DATA_BLOCK "NeuroPLC_MLP_Weights"
{ S7_Optimized_Access := 'FALSE' }
VERSION : 0.1
NON_RETAIN
   STRUCT
      w0 : ARRAY[0..895] OF REAL;  // W(32x28)
      b1 : ARRAY[0..31] OF REAL;  // bias(32)
      w2 : ARRAY[0..511] OF REAL;  // W(16x32)
      b3 : ARRAY[0..15] OF REAL;  // bias(16)
      w4 : ARRAY[0..63] OF REAL;  // W(4x16)
      b5 : ARRAY[0..3] OF REAL;  // bias(4)
   END_STRUCT;
BEGIN

      // MatMul 'fc0': W + bias
      w0[0] := 0.5694862; w0[1] := -0.0095692; w0[2] := 0.7619486; w0[3] := 0.2215109; w0[4] := -0.3561512; w0[5] := -0.2522623; w0[6] := 0.2582799; w0[7] := 0.0099258;
      w0[8] := 0.3836571; w0[9] := -0.0658457; w0[10] := 0.1010401; w0[11] := -0.2984352; w0[12] := 0.1934527; w0[13] := -0.2640140; w0[14] := 0.1362384; w0[15] := -0.0190728;
      w0[16] := -0.2375232; w0[17] := -0.1084833; w0[18] := -0.3846658; w0[19] := 0.3771667; w0[20] := -0.1136759; w0[21] := -0.1259104; w0[22] := -0.1682155; w0[23] := 0.4097499;
      w0[24] := -0.2194012; w0[25] := -0.2356472; w0[26] := -0.1771912; w0[27] := 0.1675407; w0[28] := 0.1454716; w0[29] := -0.3696787; w0[30] := -0.2783369; w0[31] := -0.1873165;
      w0[32] := 0.0781848; w0[33] := -0.3527579; w0[34] := -0.2131715; w0[35] := -0.4139680; w0[36] := -0.5927966; w0[37] := 0.3198802; w0[38] := -0.5640871; w0[39] := -0.2003005;
      w0[40] := 0.1832723; w0[41] := 0.2237836; w0[42] := 0.1929916; w0[43] := 0.2185234; w0[44] := 0.1214973; w0[45] := 0.0208249; w0[46] := 0.2776418; w0[47] := 0.6831574;
      w0[48] := -0.1655439; w0[49] := -0.2658227; w0[50] := -0.2709237; w0[51] := 0.0986710; w0[52] := 0.1128972; w0[53] := -0.2047481; w0[54] := -0.3872808; w0[55] := 0.1596099;
      w0[56] := -0.2523361; w0[57] := 0.2758174; w0[58] := 0.2686562; w0[59] := -0.5177624; w0[60] := -0.1129441; w0[61] := -0.2192100; w0[62] := 0.3343761; w0[63] := -0.0422801;
      w0[64] := -0.3068857; w0[65] := 0.2210509; w0[66] := -0.5496964; w0[67] := 0.3709493; w0[68] := 0.0747587; w0[69] := -0.1170707; w0[70] := -0.3195110; w0[71] := 0.0277475;
      w0[72] := -0.2577946; w0[73] := 0.0641775; w0[74] := 0.2055912; w0[75] := 0.6039576; w0[76] := -0.5010191; w0[77] := 0.0377836; w0[78] := 0.2038942; w0[79] := -0.0376425;
      w0[80] := 0.1546009; w0[81] := 0.3260912; w0[82] := -0.1506072; w0[83] := 0.0569262; w0[84] := -0.1928782; w0[85] := -0.1984540; w0[86] := -0.0539345; w0[87] := 0.3094364;
      w0[88] := 0.2289592; w0[89] := -0.4250050; w0[90] := -0.0399776; w0[91] := 0.0658291; w0[92] := 0.2534966; w0[93] := -0.0973715; w0[94] := -0.3647969; w0[95] := -0.0156060;
      w0[96] := -0.5209337; w0[97] := 0.2564455; w0[98] := 0.1338747; w0[99] := 0.3502659; w0[100] := -0.3756513; w0[101] := 0.2530890; w0[102] := 0.0984663; w0[103] := 0.6602526;
      w0[104] := 0.3365156; w0[105] := -0.2521311; w0[106] := 0.0946512; w0[107] := -0.6085349; w0[108] := -0.5372492; w0[109] := 0.0455726; w0[110] := -0.0786947; w0[111] := 0.0370381;
      w0[112] := -0.5858350; w0[113] := -0.7779619; w0[114] := -0.7385424; w0[115] := -0.2071060; w0[116] := 0.2831336; w0[117] := 0.3243212; w0[118] := 0.2366221; w0[119] := -0.2105746;
      w0[120] := -0.3834608; w0[121] := -0.6828474; w0[122] := 0.1007835; w0[123] := 0.0381121; w0[124] := 0.3126857; w0[125] := 0.0975034; w0[126] := 0.0499541; w0[127] := -0.0530838;
      w0[128] := 0.0799674; w0[129] := -0.1505451; w0[130] := -0.4892448; w0[131] := -0.3954702; w0[132] := 0.1594549; w0[133] := 0.2307071; w0[134] := -0.0041823; w0[135] := 0.5944483;
      w0[136] := -0.2759206; w0[137] := -0.4257804; w0[138] := -0.3279784; w0[139] := -0.2977980; w0[140] := 0.0038754; w0[141] := 0.3761657; w0[142] := 0.4177073; w0[143] := 0.0741864;
      w0[144] := 0.3750937; w0[145] := 0.2039272; w0[146] := -0.2429399; w0[147] := -0.3849822; w0[148] := 0.1600508; w0[149] := -0.1581226; w0[150] := -0.0233814; w0[151] := -0.1151747;
      w0[152] := -0.5731639; w0[153] := -0.0274457; w0[154] := 0.1195597; w0[155] := -0.2395748; w0[156] := 0.2293357; w0[157] := -0.0251415; w0[158] := 0.3937997; w0[159] := -0.1454628;
      w0[160] := -0.0673693; w0[161] := 0.2948158; w0[162] := 0.5630679; w0[163] := -0.3092144; w0[164] := 0.1832785; w0[165] := 0.0043120; w0[166] := 0.0011036; w0[167] := 0.2549984;
      w0[168] := 0.1242365; w0[169] := -0.1573328; w0[170] := 0.1472307; w0[171] := 0.2971004; w0[172] := 0.1052006; w0[173] := 0.3616425; w0[174] := -0.1347494; w0[175] := -0.3794992;
      w0[176] := 0.5467421; w0[177] := -0.1476457; w0[178] := 0.3496484; w0[179] := -0.0583753; w0[180] := 0.2853532; w0[181] := -0.3058073; w0[182] := -0.1615329; w0[183] := -0.5229150;
      w0[184] := 0.2140338; w0[185] := -0.2294949; w0[186] := 0.2921923; w0[187] := 0.0373898; w0[188] := 0.3493846; w0[189] := 0.5938788; w0[190] := 0.0955027; w0[191] := -0.1719695;
      w0[192] := 0.6582399; w0[193] := -0.4911650; w0[194] := 0.1269870; w0[195] := -0.4129370; w0[196] := -0.2735490; w0[197] := -0.2155660; w0[198] := 0.4269275; w0[199] := -0.1273027;
      w0[200] := -0.2414422; w0[201] := -0.3611139; w0[202] := 0.6480063; w0[203] := 0.3808921; w0[204] := -0.2189153; w0[205] := 0.0094489; w0[206] := 0.6784652; w0[207] := 0.3757944;
      w0[208] := 0.5965886; w0[209] := 0.3704935; w0[210] := 0.3205929; w0[211] := 0.2190031; w0[212] := -0.3913886; w0[213] := 0.2046225; w0[214] := 0.7660633; w0[215] := 0.5648795;
      w0[216] := 0.0447379; w0[217] := -0.1363681; w0[218] := -0.1653181; w0[219] := -0.3211187; w0[220] := 0.0557173; w0[221] := -0.6775630; w0[222] := 0.2077208; w0[223] := 0.1863764;
      w0[224] := 0.0122372; w0[225] := -0.1510706; w0[226] := -0.0393031; w0[227] := -0.2373850; w0[228] := 0.3297745; w0[229] := -0.3327326; w0[230] := -0.1183226; w0[231] := 0.3871697;
      w0[232] := -0.4481050; w0[233] := -0.2065133; w0[234] := 0.1012533; w0[235] := -0.2578072; w0[236] := 0.0634624; w0[237] := -0.1246978; w0[238] := 0.1465549; w0[239] := -0.5023389;
      w0[240] := 0.0640146; w0[241] := 0.1963426; w0[242] := 0.6648222; w0[243] := -0.6102669; w0[244] := -0.2871900; w0[245] := -0.3684005; w0[246] := -0.4533643; w0[247] := -0.1819637;
      w0[248] := -0.3802012; w0[249] := 0.4682154; w0[250] := 0.1991423; w0[251] := 0.5698866; w0[252] := 0.3063245; w0[253] := 0.1672625; w0[254] := 0.2611240; w0[255] := -0.6845852;
      w0[256] := -0.1005014; w0[257] := -0.6641653; w0[258] := -0.2544510; w0[259] := 0.1954752; w0[260] := -0.2994281; w0[261] := 0.3571715; w0[262] := -0.0372742; w0[263] := -0.0310561;
      w0[264] := 0.1959654; w0[265] := -0.1060541; w0[266] := 0.3827632; w0[267] := -0.3923316; w0[268] := -0.5924090; w0[269] := 0.0670658; w0[270] := 0.3532278; w0[271] := 0.6439264;
      w0[272] := 0.1193878; w0[273] := -0.5490641; w0[274] := -0.6517076; w0[275] := 0.2266813; w0[276] := 0.2735080; w0[277] := 0.2562127; w0[278] := 0.3711089; w0[279] := -0.0201157;
      w0[280] := 0.5907255; w0[281] := 0.3026478; w0[282] := 0.0879490; w0[283] := -0.1103418; w0[284] := 0.0830003; w0[285] := 0.0901832; w0[286] := 0.4872787; w0[287] := -0.4248994;
      w0[288] := 0.6916616; w0[289] := 0.0068263; w0[290] := 0.0377772; w0[291] := -0.3450460; w0[292] := 0.5848706; w0[293] := -0.0756037; w0[294] := 0.0390328; w0[295] := -0.4139087;
      w0[296] := -0.1527735; w0[297] := -0.2285863; w0[298] := 0.3310088; w0[299] := 0.2031009; w0[300] := -0.5309294; w0[301] := -0.4607368; w0[302] := 0.1824918; w0[303] := -0.1911459;
      w0[304] := -0.1732452; w0[305] := -0.3283744; w0[306] := -0.0425148; w0[307] := -0.0754750; w0[308] := -0.0751830; w0[309] := -0.0057766; w0[310] := -0.0669558; w0[311] := -0.0518108;
      w0[312] := -0.1100485; w0[313] := 0.4202482; w0[314] := 0.1722786; w0[315] := 0.2540640; w0[316] := -0.2125306; w0[317] := -0.3108644; w0[318] := -0.1653187; w0[319] := 0.0082027;
      w0[320] := 0.1613134; w0[321] := 0.5696448; w0[322] := 0.4734836; w0[323] := -0.1820288; w0[324] := -0.0202256; w0[325] := 0.2319008; w0[326] := 0.6178575; w0[327] := -0.1729726;
      w0[328] := -0.5705087; w0[329] := -0.4175466; w0[330] := -0.0846097; w0[331] := -0.4305633; w0[332] := -0.0297265; w0[333] := -0.2146564; w0[334] := -0.0228577; w0[335] := 0.4386194;
      w0[336] := 0.1366172; w0[337] := 0.1275948; w0[338] := 0.2872518; w0[339] := -0.0469490; w0[340] := -0.3430789; w0[341] := -0.2333279; w0[342] := -0.0942715; w0[343] := -0.6695372;
      w0[344] := 0.3036573; w0[345] := 0.6706407; w0[346] := 0.4867018; w0[347] := 0.2229243; w0[348] := 0.1479198; w0[349] := 0.4786703; w0[350] := -0.1235309; w0[351] := -0.1444162;
      w0[352] := -0.1594525; w0[353] := 0.0118241; w0[354] := 0.3302614; w0[355] := 0.4612524; w0[356] := -0.1728074; w0[357] := -0.4940682; w0[358] := 0.2663130; w0[359] := 0.4213447;
      w0[360] := 0.1559720; w0[361] := 0.0927116; w0[362] := 0.2581408; w0[363] := 0.1484697; w0[364] := 0.5596921; w0[365] := 0.6450443; w0[366] := 0.2316463; w0[367] := -0.3064318;
      w0[368] := 0.3154030; w0[369] := 0.2504337; w0[370] := 0.2270162; w0[371] := -0.2362736; w0[372] := -0.1822204; w0[373] := 0.7585521; w0[374] := 0.2454521; w0[375] := -0.3572387;
      w0[376] := 0.1800293; w0[377] := 0.1965537; w0[378] := 0.1946464; w0[379] := 0.1738928; w0[380] := -0.1159788; w0[381] := -0.1791228; w0[382] := 0.3109314; w0[383] := 0.1039406;
      w0[384] := -0.2558490; w0[385] := -0.4132357; w0[386] := -0.1826324; w0[387] := -0.0949509; w0[388] := 0.0754630; w0[389] := -0.4951166; w0[390] := -0.0366096; w0[391] := -0.5241205;
      w0[392] := 0.0701182; w0[393] := 0.5458165; w0[394] := -0.3082272; w0[395] := -0.1620290; w0[396] := 0.2685293; w0[397] := -0.1115321; w0[398] := 0.5528188; w0[399] := 0.1818966;
      w0[400] := -0.2705870; w0[401] := -0.4477837; w0[402] := -0.3260813; w0[403] := -0.1751753; w0[404] := 0.3439055; w0[405] := 0.3690660; w0[406] := -0.0775537; w0[407] := -0.3291571;
      w0[408] := 0.3966570; w0[409] := 0.3747428; w0[410] := 0.2037812; w0[411] := 0.5063270; w0[412] := -0.0363616; w0[413] := -0.0945516; w0[414] := -0.2667596; w0[415] := -0.1880456;
      w0[416] := 0.2148547; w0[417] := -0.6592890; w0[418] := -0.2238534; w0[419] := -0.2862469; w0[420] := -0.8308039; w0[421] := -0.4430834; w0[422] := -0.0302747; w0[423] := 0.0918460;
      w0[424] := -0.3334551; w0[425] := -0.1804388; w0[426] := -0.1097601; w0[427] := 0.3427432; w0[428] := 0.0736062; w0[429] := -0.6790179; w0[430] := -0.2430520; w0[431] := -0.2084594;
      w0[432] := 0.1491454; w0[433] := -0.0083196; w0[434] := 0.2553293; w0[435] := 0.1678275; w0[436] := 0.0936099; w0[437] := 0.1736043; w0[438] := -0.5376837; w0[439] := -0.4510113;
      w0[440] := -0.3174161; w0[441] := 0.2371299; w0[442] := 0.3883051; w0[443] := 0.3464468; w0[444] := 0.1098732; w0[445] := 0.0205052; w0[446] := -0.2641115; w0[447] := -0.3012585;
      w0[448] := -0.5463231; w0[449] := -0.0684724; w0[450] := -0.1422806; w0[451] := -0.2644515; w0[452] := -0.4767578; w0[453] := -0.4182616; w0[454] := -0.4673964; w0[455] := -0.0129319;
      w0[456] := -0.5374129; w0[457] := -0.1050398; w0[458] := 0.0632549; w0[459] := 0.0568505; w0[460] := 0.2111508; w0[461] := 0.3917949; w0[462] := -0.0330271; w0[463] := 0.2814879;
      w0[464] := -0.3214771; w0[465] := 0.3430510; w0[466] := -0.3870021; w0[467] := -0.4042188; w0[468] := 0.1747253; w0[469] := 0.3262924; w0[470] := 0.5594077; w0[471] := 0.0277393;
      w0[472] := -0.2604083; w0[473] := 0.0503597; w0[474] := 0.3725081; w0[475] := -0.0544451; w0[476] := 0.0951887; w0[477] := -0.5271522; w0[478] := -0.3720489; w0[479] := 0.0333015;
      w0[480] := 0.3407656; w0[481] := -0.0524092; w0[482] := -0.3947720; w0[483] := 0.0632993; w0[484] := -0.4918242; w0[485] := -0.0408889; w0[486] := 0.5603451; w0[487] := 0.3429145;
      w0[488] := -0.0672607; w0[489] := -0.3218429; w0[490] := -0.3621323; w0[491] := -0.5524946; w0[492] := 0.3105496; w0[493] := 0.3352183; w0[494] := -0.6259544; w0[495] := -0.1107638;
      w0[496] := 0.0901521; w0[497] := 0.0038500; w0[498] := 0.5420415; w0[499] := 0.2380718; w0[500] := -0.0511688; w0[501] := -0.0771460; w0[502] := -0.0791493; w0[503] := -0.1069665;
      w0[504] := 0.6399192; w0[505] := -0.0014034; w0[506] := 0.3290343; w0[507] := -0.3565734; w0[508] := 0.2305476; w0[509] := -0.0417552; w0[510] := 0.2942790; w0[511] := -0.1355964;
      w0[512] := 0.0557771; w0[513] := 0.3271682; w0[514] := -0.3025698; w0[515] := 0.2897500; w0[516] := 0.1278277; w0[517] := -0.1560617; w0[518] := 0.2582703; w0[519] := -0.0549245;
      w0[520] := -0.0921321; w0[521] := 0.4996554; w0[522] := 0.0836308; w0[523] := 0.2032579; w0[524] := -0.1741465; w0[525] := -0.2436171; w0[526] := -0.3661414; w0[527] := -0.2924559;
      w0[528] := -0.4407195; w0[529] := 0.2304931; w0[530] := -0.2509898; w0[531] := -0.6881460; w0[532] := 0.1500384; w0[533] := 0.4429501; w0[534] := 0.5444623; w0[535] := 0.0644146;
      w0[536] := 0.1564979; w0[537] := 0.1936211; w0[538] := -0.2217757; w0[539] := 0.1632960; w0[540] := 0.0949209; w0[541] := 0.5449093; w0[542] := 0.3260632; w0[543] := 0.4177442;
      w0[544] := -0.1678705; w0[545] := -0.4614883; w0[546] := -0.1780888; w0[547] := 0.0282706; w0[548] := -0.3548764; w0[549] := 0.1119965; w0[550] := -0.6278588; w0[551] := -0.2857478;
      w0[552] := 0.3291071; w0[553] := -0.2958602; w0[554] := -0.2171935; w0[555] := 0.0488607; w0[556] := -0.2721503; w0[557] := -0.0109805; w0[558] := -0.2872001; w0[559] := -0.3800366;
      w0[560] := 0.7377275; w0[561] := 0.5175216; w0[562] := 0.4534726; w0[563] := 0.2131705; w0[564] := 0.1694544; w0[565] := 0.1088488; w0[566] := 0.2956495; w0[567] := -0.1219863;
      w0[568] := 0.4281839; w0[569] := 0.0482728; w0[570] := 0.3261450; w0[571] := 0.0147065; w0[572] := 0.0197347; w0[573] := -0.2837075; w0[574] := -0.2223815; w0[575] := -0.3011971;
      w0[576] := 0.4010099; w0[577] := 0.3606303; w0[578] := 0.5675586; w0[579] := -0.1933776; w0[580] := 0.1411208; w0[581] := 0.4412328; w0[582] := -0.3157989; w0[583] := 0.0737199;
      w0[584] := 0.2547267; w0[585] := -0.4104514; w0[586] := 0.3333948; w0[587] := 0.0244799; w0[588] := 0.3485871; w0[589] := -0.1856655; w0[590] := -0.2338329; w0[591] := -0.2214157;
      w0[592] := 0.4647014; w0[593] := -0.3053385; w0[594] := -0.1758788; w0[595] := -0.2062785; w0[596] := 0.4421045; w0[597] := 0.2903270; w0[598] := 0.2819436; w0[599] := -0.3433319;
      w0[600] := -0.0214767; w0[601] := 0.5416198; w0[602] := -0.0143610; w0[603] := -0.1832658; w0[604] := -0.5633022; w0[605] := -0.1308155; w0[606] := 0.1253684; w0[607] := -0.3460040;
      w0[608] := -0.0773746; w0[609] := -0.0179889; w0[610] := -0.3036036; w0[611] := 0.0990553; w0[612] := -0.2073587; w0[613] := 0.0275394; w0[614] := 0.0471204; w0[615] := -0.0187443;
      w0[616] := 0.4038751; w0[617] := 0.0922068; w0[618] := -0.2135524; w0[619] := -0.4082574; w0[620] := -0.0358560; w0[621] := -0.1610684; w0[622] := -0.4163499; w0[623] := 0.2467240;
      w0[624] := 0.0747931; w0[625] := 0.3987921; w0[626] := 0.1632655; w0[627] := -0.3848493; w0[628] := 0.1649167; w0[629] := -0.6442378; w0[630] := -0.4510081; w0[631] := -0.2822698;
      w0[632] := 0.4664556; w0[633] := -0.2991767; w0[634] := -0.0362801; w0[635] := -0.3327457; w0[636] := -0.3074295; w0[637] := 0.1606831; w0[638] := -0.0541677; w0[639] := -0.5748461;
      w0[640] := 0.3949239; w0[641] := -0.2336025; w0[642] := -0.0525538; w0[643] := 0.3131756; w0[644] := -0.0032524; w0[645] := -0.0003879; w0[646] := 0.3644529; w0[647] := 0.3278647;
      w0[648] := -0.0496909; w0[649] := -0.0200011; w0[650] := 0.4739185; w0[651] := -0.3886660; w0[652] := 0.0855980; w0[653] := -0.4665208; w0[654] := 0.4008028; w0[655] := -0.5448800;
      w0[656] := -0.4093939; w0[657] := -0.1329360; w0[658] := 0.2988919; w0[659] := -0.0788539; w0[660] := 0.0282110; w0[661] := -0.1015701; w0[662] := 0.5736219; w0[663] := -0.2615215;
      w0[664] := 0.0237927; w0[665] := 0.0321014; w0[666] := -0.1239056; w0[667] := -0.2004481; w0[668] := -0.0194097; w0[669] := -0.1323835; w0[670] := -0.0777957; w0[671] := 0.0366594;
      w0[672] := 0.1079154; w0[673] := 0.4157223; w0[674] := -0.2902254; w0[675] := 0.4283061; w0[676] := 0.0650300; w0[677] := 0.1249261; w0[678] := -0.2917063; w0[679] := -0.1270394;
      w0[680] := 0.0782463; w0[681] := 0.5982807; w0[682] := 0.1017760; w0[683] := 0.1843081; w0[684] := -0.6125457; w0[685] := 0.2722199; w0[686] := -0.0728571; w0[687] := -0.5004624;
      w0[688] := 0.4432183; w0[689] := 0.4912130; w0[690] := 0.0002442; w0[691] := -0.0942999; w0[692] := 0.5940161; w0[693] := -0.1235101; w0[694] := 0.3478113; w0[695] := 0.0345737;
      w0[696] := -0.0406947; w0[697] := 0.6151400; w0[698] := 0.2030335; w0[699] := -0.3236780; w0[700] := -0.6019017; w0[701] := -0.4779230; w0[702] := -0.8101817; w0[703] := -0.2094196;
      w0[704] := -0.3149875; w0[705] := 0.3055148; w0[706] := -0.2818980; w0[707] := 0.2800311; w0[708] := -0.8234739; w0[709] := -0.6584272; w0[710] := 0.2585062; w0[711] := 0.0584044;
      w0[712] := -0.5591815; w0[713] := -0.0547792; w0[714] := 0.0355113; w0[715] := 0.2701355; w0[716] := -0.5936313; w0[717] := 0.3193162; w0[718] := 0.1195579; w0[719] := 0.0537417;
      w0[720] := 0.6140408; w0[721] := 0.5008627; w0[722] := -0.0104372; w0[723] := 0.2329175; w0[724] := -0.0168664; w0[725] := 0.0332739; w0[726] := 0.3730388; w0[727] := 0.1635417;
      w0[728] := 0.7335413; w0[729] := 0.5691491; w0[730] := 0.0170918; w0[731] := 0.2825087; w0[732] := 0.0198349; w0[733] := 0.4498756; w0[734] := 0.4100120; w0[735] := -0.2479021;
      w0[736] := 0.2850291; w0[737] := -0.1702987; w0[738] := -0.4980538; w0[739] := -0.0941117; w0[740] := 0.4272463; w0[741] := -0.2824812; w0[742] := 0.6535753; w0[743] := 0.2375765;
      w0[744] := 0.4509313; w0[745] := -0.0013205; w0[746] := 0.1127060; w0[747] := -0.1239916; w0[748] := 0.3028973; w0[749] := 0.0927592; w0[750] := -0.3168923; w0[751] := 0.1611173;
      w0[752] := 0.4917028; w0[753] := 0.0417323; w0[754] := 0.3917417; w0[755] := -0.0557213; w0[756] := -0.2345485; w0[757] := 0.3833969; w0[758] := 0.3747815; w0[759] := -0.1519468;
      w0[760] := -0.3892233; w0[761] := -0.0699942; w0[762] := -0.3351573; w0[763] := -0.3026012; w0[764] := -0.1781991; w0[765] := 0.4689204; w0[766] := -0.1804391; w0[767] := -0.2284776;
      w0[768] := -0.3932275; w0[769] := 0.2445571; w0[770] := -0.1087966; w0[771] := -0.2825441; w0[772] := -0.2301650; w0[773] := 0.5091258; w0[774] := -0.7006359; w0[775] := 0.0339814;
      w0[776] := 0.1417895; w0[777] := 0.1839303; w0[778] := 0.2910166; w0[779] := 0.1044962; w0[780] := 0.0580844; w0[781] := 0.6158280; w0[782] := -0.0284938; w0[783] := 0.0542879;
      w0[784] := 0.1680317; w0[785] := 0.2264472; w0[786] := -0.2030084; w0[787] := 0.0756811; w0[788] := -0.2188872; w0[789] := -0.2264328; w0[790] := -0.1813061; w0[791] := -0.2645762;
      w0[792] := 0.4621922; w0[793] := -0.4514092; w0[794] := 0.3058094; w0[795] := 0.3434274; w0[796] := 0.3808913; w0[797] := -0.3231871; w0[798] := 0.2469297; w0[799] := -0.1890893;
      w0[800] := 0.0499585; w0[801] := -0.3218643; w0[802] := 0.6025205; w0[803] := 0.0650566; w0[804] := -0.2298092; w0[805] := 0.5071256; w0[806] := -0.2657916; w0[807] := -0.1830709;
      w0[808] := 0.0415640; w0[809] := -0.1594847; w0[810] := -0.0321660; w0[811] := -0.0346579; w0[812] := -0.3819390; w0[813] := 0.2074234; w0[814] := 0.3919429; w0[815] := 0.0324158;
      w0[816] := -0.0215873; w0[817] := -0.1329270; w0[818] := 0.0735578; w0[819] := 0.3148956; w0[820] := -0.4435450; w0[821] := -0.3320747; w0[822] := -0.1767979; w0[823] := -0.4104172;
      w0[824] := 0.3253109; w0[825] := -0.1773608; w0[826] := -0.4930988; w0[827] := 0.3281353; w0[828] := 0.3916833; w0[829] := -0.1541856; w0[830] := 0.1263307; w0[831] := 0.0426248;
      w0[832] := -0.5533415; w0[833] := 0.0726361; w0[834] := -0.4881184; w0[835] := -0.1073755; w0[836] := -0.5946367; w0[837] := -0.5742470; w0[838] := 0.1233901; w0[839] := -0.0872265;
      w0[840] := 0.2010813; w0[841] := 0.4012275; w0[842] := 0.3290967; w0[843] := 0.3005436; w0[844] := -0.0111396; w0[845] := -0.4794478; w0[846] := -0.0532993; w0[847] := -0.1733176;
      w0[848] := -0.1260332; w0[849] := 0.1089438; w0[850] := 0.0391418; w0[851] := -0.2468968; w0[852] := 0.4689822; w0[853] := -0.4640872; w0[854] := 0.2532913; w0[855] := -0.2343228;
      w0[856] := 0.2661497; w0[857] := -0.4386278; w0[858] := 0.0468966; w0[859] := -0.3265733; w0[860] := -0.1916417; w0[861] := 0.5178355; w0[862] := 0.2822486; w0[863] := -0.1077720;
      w0[864] := 0.3286300; w0[865] := -0.0029810; w0[866] := -0.3535745; w0[867] := -0.1011055; w0[868] := 0.1318278; w0[869] := 0.0674391; w0[870] := 0.0591611; w0[871] := -0.1122496;
      w0[872] := 0.4686061; w0[873] := -0.4002847; w0[874] := 0.0749937; w0[875] := -0.1933431; w0[876] := 0.2702274; w0[877] := -0.1278288; w0[878] := -0.1761822; w0[879] := -0.2737747;
      w0[880] := 0.4466998; w0[881] := 0.0271071; w0[882] := 0.1916832; w0[883] := 0.4834492; w0[884] := 0.0259246; w0[885] := -0.4892190; w0[886] := 0.2059345; w0[887] := -0.0822330;
      w0[888] := -0.4142632; w0[889] := 0.5404200; w0[890] := -0.1093403; w0[891] := 0.0186543; w0[892] := 0.6250578; w0[893] := -0.2241697; w0[894] := 0.3088920; w0[895] := 0.1112378;
      b1[0] := -0.1609981; b1[1] := -0.0371174; b1[2] := 0.0221225; b1[3] := 0.0337845; b1[4] := 0.2616802; b1[5] := 0.1264098; b1[6] := 0.1833381; b1[7] := 0.1271529;
      b1[8] := 0.0488858; b1[9] := 0.0241906; b1[10] := -0.3121075; b1[11] := 0.0973287; b1[12] := -0.0882614; b1[13] := -0.3344531; b1[14] := -0.1306882; b1[15] := 0.1518650;
      b1[16] := 0.0104939; b1[17] := -0.0685202; b1[18] := -0.0953050; b1[19] := 0.0008646; b1[20] := 0.2513834; b1[21] := 0.0002911; b1[22] := 0.1923783; b1[23] := 0.1726166;
      b1[24] := 0.3154603; b1[25] := 0.0885571; b1[26] := 0.0390019; b1[27] := 0.0755870; b1[28] := 0.1380671; b1[29] := 0.1447226; b1[30] := 0.0485010; b1[31] := 0.1450995;

      // MatMul 'fc1': W + bias
      w2[0] := 0.3448875; w2[1] := -0.0985299; w2[2] := -0.2385274; w2[3] := 0.1068773; w2[4] := 0.5171419; w2[5] := -0.1054032; w2[6] := 0.2936411; w2[7] := -0.4853331;
      w2[8] := -0.3005029; w2[9] := 0.2366145; w2[10] := 0.3783182; w2[11] := 0.1278910; w2[12] := 0.0211917; w2[13] := -0.1069832; w2[14] := -0.2683547; w2[15] := -0.0976455;
      w2[16] := 0.6765909; w2[17] := 0.5036446; w2[18] := 0.3599868; w2[19] := 0.0810751; w2[20] := -0.0792580; w2[21] := -0.2718676; w2[22] := -0.4316851; w2[23] := -0.1867653;
      w2[24] := 0.2037492; w2[25] := -0.0189868; w2[26] := -0.0119788; w2[27] := 0.3331117; w2[28] := -0.1736732; w2[29] := -0.4839838; w2[30] := -0.0297980; w2[31] := -0.6352752;
      w2[32] := 0.4027197; w2[33] := -0.5263022; w2[34] := 0.2703936; w2[35] := 0.1180763; w2[36] := -0.3752257; w2[37] := -0.6156019; w2[38] := -0.4087748; w2[39] := 0.1517635;
      w2[40] := 0.2814839; w2[41] := -0.3188637; w2[42] := 0.4876765; w2[43] := 0.1747880; w2[44] := -0.1799005; w2[45] := -0.3207765; w2[46] := 0.6545156; w2[47] := -0.3893254;
      w2[48] := -0.3369366; w2[49] := -0.4376430; w2[50] := 0.0413780; w2[51] := -0.1731163; w2[52] := 0.3791941; w2[53] := 0.0461393; w2[54] := 0.0816816; w2[55] := 0.3956819;
      w2[56] := -0.3843228; w2[57] := -0.7061806; w2[58] := -0.6190179; w2[59] := -0.4308152; w2[60] := 0.2132129; w2[61] := 0.4490756; w2[62] := -0.2397823; w2[63] := 0.3091693;
      w2[64] := -0.1736172; w2[65] := -0.6044765; w2[66] := 0.2081352; w2[67] := 0.4768652; w2[68] := -0.2759739; w2[69] := 0.1133698; w2[70] := -0.0100859; w2[71] := -0.6772556;
      w2[72] := 0.5169631; w2[73] := 0.1017481; w2[74] := -0.0672581; w2[75] := -0.4697476; w2[76] := -0.1098660; w2[77] := -0.1401970; w2[78] := -0.4618214; w2[79] := -0.2387714;
      w2[80] := -0.3492894; w2[81] := -0.2289385; w2[82] := 0.3859353; w2[83] := 0.3484918; w2[84] := 0.0570800; w2[85] := 0.4838708; w2[86] := 0.4412340; w2[87] := 0.1156965;
      w2[88] := 0.4213234; w2[89] := -0.2558614; w2[90] := 0.2997079; w2[91] := -0.0041088; w2[92] := -0.2610477; w2[93] := -0.2681805; w2[94] := 0.7025032; w2[95] := 0.4033620;
      w2[96] := 0.0018223; w2[97] := 0.3965206; w2[98] := -0.1132530; w2[99] := 0.3405365; w2[100] := 0.4333419; w2[101] := 0.0468351; w2[102] := -0.4313038; w2[103] := -0.5938676;
      w2[104] := -0.1057017; w2[105] := 0.3874305; w2[106] := -0.3047897; w2[107] := -0.3605830; w2[108] := -0.0865778; w2[109] := 0.0169620; w2[110] := -0.2818013; w2[111] := -0.2056310;
      w2[112] := 0.2889744; w2[113] := -0.2389124; w2[114] := -0.5219849; w2[115] := -0.5379763; w2[116] := -0.3595321; w2[117] := 0.2131797; w2[118] := 0.2746126; w2[119] := 0.2555465;
      w2[120] := -0.3816569; w2[121] := -0.1742714; w2[122] := -0.3458711; w2[123] := -0.4732965; w2[124] := 0.3816739; w2[125] := 0.4522255; w2[126] := 0.4340182; w2[127] := 0.1317699;
      w2[128] := 0.0887004; w2[129] := -0.1704083; w2[130] := 0.2312619; w2[131] := -0.1512796; w2[132] := 0.1522121; w2[133] := -0.3580639; w2[134] := 0.3120518; w2[135] := -0.0891345;
      w2[136] := -0.5189782; w2[137] := 0.6759704; w2[138] := 0.8410841; w2[139] := -0.4388631; w2[140] := 0.3120123; w2[141] := 0.0530660; w2[142] := -0.1540236; w2[143] := -0.1420563;
      w2[144] := 0.3882907; w2[145] := 0.3881267; w2[146] := 0.4476533; w2[147] := 0.4830106; w2[148] := 0.2335594; w2[149] := 0.1241002; w2[150] := -0.2032309; w2[151] := -0.5769788;
      w2[152] := 0.3601961; w2[153] := 0.5940281; w2[154] := -0.3626602; w2[155] := 0.1981693; w2[156] := -0.0685700; w2[157] := -0.0704796; w2[158] := 0.0195035; w2[159] := -0.4674689;
      w2[160] := -0.2348353; w2[161] := -0.3250483; w2[162] := 0.1978887; w2[163] := -0.0533809; w2[164] := 0.5541837; w2[165] := 0.0647560; w2[166] := 0.1574209; w2[167] := -0.4176951;
      w2[168] := -0.0328900; w2[169] := -0.4697271; w2[170] := -0.0496295; w2[171] := -0.1912494; w2[172] := -0.2456453; w2[173] := -0.3518490; w2[174] := 0.0067706; w2[175] := 0.6691334;
      w2[176] := 0.5995317; w2[177] := 0.3372136; w2[178] := -0.2781896; w2[179] := 0.2096184; w2[180] := -0.4983254; w2[181] := -0.0787928; w2[182] := -0.2063265; w2[183] := -0.2567849;
      w2[184] := -0.2985751; w2[185] := 0.2627156; w2[186] := 0.1459312; w2[187] := 0.4578165; w2[188] := 0.0136775; w2[189] := 0.4329558; w2[190] := -0.2819005; w2[191] := 0.0772760;
      w2[192] := 0.1485205; w2[193] := 0.0424627; w2[194] := -0.5533946; w2[195] := -0.3114872; w2[196] := -0.0971009; w2[197] := 0.1043289; w2[198] := -0.0080725; w2[199] := 0.0561389;
      w2[200] := 0.1712011; w2[201] := -0.2093053; w2[202] := -0.4844932; w2[203] := 0.5200891; w2[204] := -0.4811763; w2[205] := -0.2097965; w2[206] := -0.1644997; w2[207] := 0.0035760;
      w2[208] := 0.2773729; w2[209] := 0.4809147; w2[210] := -0.3132524; w2[211] := -0.0345517; w2[212] := 0.5111094; w2[213] := 0.1451371; w2[214] := 0.0575851; w2[215] := 0.1672285;
      w2[216] := 0.3724994; w2[217] := 0.0500904; w2[218] := -0.0895519; w2[219] := 0.0279228; w2[220] := -0.0756062; w2[221] := -0.6023685; w2[222] := 0.5966649; w2[223] := -0.4288191;
      w2[224] := -0.2491551; w2[225] := 0.1842164; w2[226] := 0.1995990; w2[227] := 0.3348442; w2[228] := -0.6874152; w2[229] := 0.0923893; w2[230] := 0.5566139; w2[231] := 0.6076588;
      w2[232] := 0.4055642; w2[233] := 0.1035502; w2[234] := -0.2282035; w2[235] := 0.0315236; w2[236] := 0.3474000; w2[237] := 0.1027276; w2[238] := 0.0550077; w2[239] := -0.1958367;
      w2[240] := -0.1637788; w2[241] := 0.2277053; w2[242] := -0.1716563; w2[243] := 0.1922517; w2[244] := 0.2188656; w2[245] := 0.0905953; w2[246] := -0.2237651; w2[247] := 0.4562837;
      w2[248] := -0.4297628; w2[249] := 0.0540233; w2[250] := -0.2155596; w2[251] := -0.4905677; w2[252] := 0.2578664; w2[253] := -0.0752592; w2[254] := 0.3203000; w2[255] := 0.2922962;
      w2[256] := 0.6623323; w2[257] := -0.2237271; w2[258] := -0.3789170; w2[259] := -0.3014932; w2[260] := 0.3499548; w2[261] := -0.3618023; w2[262] := -0.1381309; w2[263] := -0.2487616;
      w2[264] := -0.2042618; w2[265] := -0.3798007; w2[266] := 0.2168026; w2[267] := -0.5617495; w2[268] := 0.5470159; w2[269] := 0.3855161; w2[270] := -0.1744407; w2[271] := -0.0063227;
      w2[272] := -0.0175713; w2[273] := 0.4657946; w2[274] := 0.2311470; w2[275] := 0.2995405; w2[276] := -0.2337339; w2[277] := 0.2714463; w2[278] := -0.1801859; w2[279] := -0.2387183;
      w2[280] := 0.2680195; w2[281] := 0.4208193; w2[282] := 0.0763752; w2[283] := -0.0259924; w2[284] := -0.5796329; w2[285] := -0.4459113; w2[286] := -0.0650182; w2[287] := 0.0992380;
      w2[288] := -0.2287219; w2[289] := 0.1592736; w2[290] := 0.2655782; w2[291] := -0.7133095; w2[292] := -0.0750051; w2[293] := 0.1930008; w2[294] := 0.2515846; w2[295] := -0.1046810;
      w2[296] := 0.3638516; w2[297] := -0.5185701; w2[298] := -0.1378490; w2[299] := 0.1176404; w2[300] := -0.1728815; w2[301] := -0.4648141; w2[302] := -0.0106897; w2[303] := 0.2669196;
      w2[304] := -0.2057847; w2[305] := -0.0459625; w2[306] := -0.0872513; w2[307] := -0.5442434; w2[308] := 0.4806913; w2[309] := -0.2794292; w2[310] := 0.6181495; w2[311] := 0.4071167;
      w2[312] := -0.3071254; w2[313] := 0.1203253; w2[314] := 0.3505305; w2[315] := -0.5886531; w2[316] := -0.2951987; w2[317] := 0.3731146; w2[318] := 0.2878209; w2[319] := 0.2473200;
      w2[320] := -0.1784255; w2[321] := 0.4152616; w2[322] := 0.5053530; w2[323] := 0.2126275; w2[324] := 0.3228098; w2[325] := -0.3918779; w2[326] := -0.1658438; w2[327] := 0.5003296;
      w2[328] := -0.0053924; w2[329] := 0.0667791; w2[330] := 0.4097935; w2[331] := 0.1006095; w2[332] := 0.6046916; w2[333] := -0.0676274; w2[334] := -0.1915504; w2[335] := 0.3883604;
      w2[336] := 0.4911340; w2[337] := 0.5468511; w2[338] := -0.1983627; w2[339] := -0.0676885; w2[340] := -0.3710055; w2[341] := 0.1606412; w2[342] := 0.4564988; w2[343] := -0.5501073;
      w2[344] := -0.1039538; w2[345] := -0.0296496; w2[346] := -0.5341417; w2[347] := -0.2000433; w2[348] := 0.2511403; w2[349] := 0.3043574; w2[350] := -0.1509714; w2[351] := 0.4652316;
      w2[352] := 0.5162573; w2[353] := -0.4559039; w2[354] := 0.1557730; w2[355] := -0.3858083; w2[356] := 0.0727105; w2[357] := -0.4605626; w2[358] := -0.0643399; w2[359] := -0.2012528;
      w2[360] := -0.2376907; w2[361] := 0.6337410; w2[362] := 0.7189264; w2[363] := 0.2091954; w2[364] := 0.7626936; w2[365] := 0.3527288; w2[366] := -0.1358239; w2[367] := 0.3472250;
      w2[368] := -0.0854939; w2[369] := 0.3039412; w2[370] := 0.2409862; w2[371] := 0.4435183; w2[372] := 0.4328762; w2[373] := -0.0231600; w2[374] := -0.1171540; w2[375] := 0.0108573;
      w2[376] := -0.0911193; w2[377] := -0.5950353; w2[378] := -0.1391228; w2[379] := 0.1307337; w2[380] := -0.1149503; w2[381] := -0.0330209; w2[382] := -0.4081971; w2[383] := -0.3619282;
      w2[384] := -0.1067709; w2[385] := -0.0438268; w2[386] := 0.1861137; w2[387] := 0.1071503; w2[388] := -0.6722144; w2[389] := 0.5858943; w2[390] := 0.1327110; w2[391] := 0.3459137;
      w2[392] := 0.3487434; w2[393] := 0.0373104; w2[394] := -0.2565190; w2[395] := 0.4223759; w2[396] := -0.2403768; w2[397] := -0.0137525; w2[398] := 0.1307058; w2[399] := -0.5750338;
      w2[400] := -0.6017820; w2[401] := 0.1216069; w2[402] := -0.0930582; w2[403] := 0.0528917; w2[404] := 0.2642088; w2[405] := 0.1213500; w2[406] := -0.0773624; w2[407] := 0.1509228;
      w2[408] := 0.1637788; w2[409] := -0.0275139; w2[410] := 0.5865979; w2[411] := -0.2206961; w2[412] := 0.5099282; w2[413] := 0.2631257; w2[414] := 0.4237445; w2[415] := 0.4448525;
      w2[416] := 0.4446503; w2[417] := 0.0053865; w2[418] := -0.5579309; w2[419] := -0.1395655; w2[420] := -0.1579983; w2[421] := -0.3564516; w2[422] := 0.0891758; w2[423] := 0.1217025;
      w2[424] := -0.3250042; w2[425] := -0.0731721; w2[426] := 0.5731527; w2[427] := 0.3349074; w2[428] := -0.2764013; w2[429] := 0.3669565; w2[430] := 0.1658501; w2[431] := -0.0952915;
      w2[432] := 0.1848216; w2[433] := -0.3777516; w2[434] := 0.4125981; w2[435] := -0.2243889; w2[436] := 0.2011978; w2[437] := 0.3032005; w2[438] := 0.0724154; w2[439] := 0.2386405;
      w2[440] := -0.4659944; w2[441] := -0.5817581; w2[442] := -0.3680228; w2[443] := -0.5429725; w2[444] := -0.4282436; w2[445] := -0.0057439; w2[446] := 0.1407171; w2[447] := -0.0961595;
      w2[448] := -0.0304086; w2[449] := -0.5598830; w2[450] := -0.5288109; w2[451] := 0.2501028; w2[452] := -0.1907448; w2[453] := 0.3364898; w2[454] := 0.3753116; w2[455] := -0.1153062;
      w2[456] := -0.0149126; w2[457] := -0.3870158; w2[458] := -0.1154010; w2[459] := 0.0744122; w2[460] := -0.4487402; w2[461] := -0.2563244; w2[462] := 0.0335258; w2[463] := -0.1682583;
      w2[464] := 0.0443628; w2[465] := 0.3070406; w2[466] := -0.0503107; w2[467] := 0.0992935; w2[468] := 0.5251856; w2[469] := 0.6111719; w2[470] := 0.6419194; w2[471] := 0.1297791;
      w2[472] := 0.1860752; w2[473] := -0.1274762; w2[474] := 0.3434472; w2[475] := 0.5505610; w2[476] := 0.3397494; w2[477] := -0.5685602; w2[478] := 0.0005795; w2[479] := -0.1080624;
      w2[480] := 0.3114881; w2[481] := 0.4475129; w2[482] := 0.1615055; w2[483] := -0.4390773; w2[484] := -0.0133804; w2[485] := -0.3265319; w2[486] := -0.5983120; w2[487] := -0.2533576;
      w2[488] := 0.2004646; w2[489] := -0.2516977; w2[490] := -0.2211783; w2[491] := -0.0643062; w2[492] := 0.1233937; w2[493] := 0.1260124; w2[494] := -0.2689813; w2[495] := 0.3791626;
      w2[496] := 0.3063162; w2[497] := -0.2886556; w2[498] := -0.1805890; w2[499] := -0.1727612; w2[500] := -0.2364416; w2[501] := -0.0335479; w2[502] := 0.1661869; w2[503] := 0.1447821;
      w2[504] := -0.1905543; w2[505] := -0.4342808; w2[506] := -0.0012427; w2[507] := -0.4948293; w2[508] := 0.0922625; w2[509] := 0.0781584; w2[510] := 0.4070034; w2[511] := 0.0575855;
      b3[0] := -0.0313972; b3[1] := -0.1867536; b3[2] := 0.2673712; b3[3] := 0.0710777; b3[4] := -0.2155338; b3[5] := 0.0103840; b3[6] := 0.4061291; b3[7] := -0.0612305;
      b3[8] := 0.0899094; b3[9] := 0.1921517; b3[10] := 0.1069144; b3[11] := -0.0515455; b3[12] := 0.1089574; b3[13] := -0.1325741; b3[14] := 0.2726102; b3[15] := 0.1574048;

      // MatMul 'fc2': W + bias
      w4[0] := -0.0865753; w4[1] := -0.5062438; w4[2] := 0.1554476; w4[3] := 0.7071172; w4[4] := -0.1023560; w4[5] := 0.5811852; w4[6] := -0.6674285; w4[7] := -0.6164539;
      w4[8] := -0.8109480; w4[9] := 0.6379222; w4[10] := 0.3449526; w4[11] := -0.0613255; w4[12] := -0.0052660; w4[13] := -0.7050505; w4[14] := -0.6678494; w4[15] := 0.7979829;
      w4[16] := -0.0429653; w4[17] := -0.3721911; w4[18] := 0.9616893; w4[19] := -0.2787606; w4[20] := -0.1421925; w4[21] := -0.1321686; w4[22] := 0.1806948; w4[23] := -0.1417111;
      w4[24] := -0.4919258; w4[25] := 0.7062184; w4[26] := -0.4885310; w4[27] := -0.5391713; w4[28] := 0.7159519; w4[29] := -0.5416421; w4[30] := 0.8190475; w4[31] := -0.2587632;
      w4[32] := 0.7209747; w4[33] := -0.5606546; w4[34] := 0.2996863; w4[35] := -0.4360698; w4[36] := 0.6557293; w4[37] := 0.7114502; w4[38] := -0.0711865; w4[39] := -0.5944882;
      w4[40] := 0.5009670; w4[41] := -0.2733661; w4[42] := 0.0057439; w4[43] := 0.7727029; w4[44] := -0.5340657; w4[45] := 0.0551448; w4[46] := 0.2726173; w4[47] := -0.4893947;
      w4[48] := 0.2866370; w4[49] := 0.6904863; w4[50] := -0.7133542; w4[51] := 0.1576146; w4[52] := 0.5721015; w4[53] := 0.0582882; w4[54] := -0.7719719; w4[55] := 0.2141585;
      w4[56] := -0.2926230; w4[57] := -0.4390040; w4[58] := 0.2077623; w4[59] := 0.5338089; w4[60] := 0.5839869; w4[61] := 0.7652564; w4[62] := -0.3743652; w4[63] := -0.1907377;
      b5[0] := -0.1430807; b5[1] := 0.2929625; b5[2] := 0.1342851; b5[3] := -0.1236853;

END_DATA_BLOCK
